(* PLC project sample_project, sample_company sample_product 1 *)
(* stored: creationDateTime 2024-07-18T21:30:47, modificationDateTime 2024-07-18T22:03:54 *)

FUNCTION_BLOCK sample_function_block_FBD
  VAR_INPUT
    Reset : BOOL;
  END_VAR
  VAR_OUTPUT
    Out : INT;
  END_VAR
  VAR
    Cnt : INT;
  END_VAR
  VAR_EXTERNAL CONSTANT
    ResetCounterValue : INT;
  END_VAR
  VAR  (* added by the conversion: wires and edge detectors of the diagram *)
    _SEL4_OUT : ANY;
  END_VAR

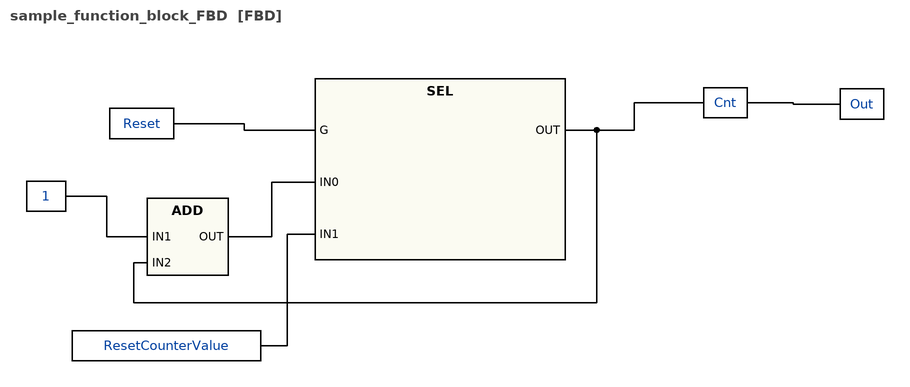
(* FBD diagram, written out as Structured Text *)
Out := Cnt;
_SEL4_OUT := SEL(Reset, 1 + _SEL4_OUT, ResetCounterValue);
Cnt := _SEL4_OUT;
END_FUNCTION_BLOCK

(* Counter in ST language *)
FUNCTION_BLOCK sample_function_block_ST
  VAR_INPUT
    Reset : BOOL;
  END_VAR
  VAR_OUTPUT
    Out : INT;
  END_VAR
  VAR
    Cnt : INT;
  END_VAR
  VAR_EXTERNAL CONSTANT
    ResetCounterValue : INT;
  END_VAR

            IF Reset THEN
  Cnt := ResetCounterValue;
ELSE
  Cnt := Cnt + 1;
END_IF;

Out := Cnt;
          
END_FUNCTION_BLOCK

PROGRAM sample_program
  VAR_INPUT
    Reset : BOOL;
  END_VAR
  VAR_OUTPUT
    Cnt0 : INT;
    Cnt1 : INT;
    Cnt2 : INT;
    Cnt3 : INT;
    Cnt4 : INT;
  END_VAR
  VAR
    sample_function_block_ST0 : sample_function_block_ST;
    sample_function_block_FBD0 : sample_function_block_FBD;
  END_VAR

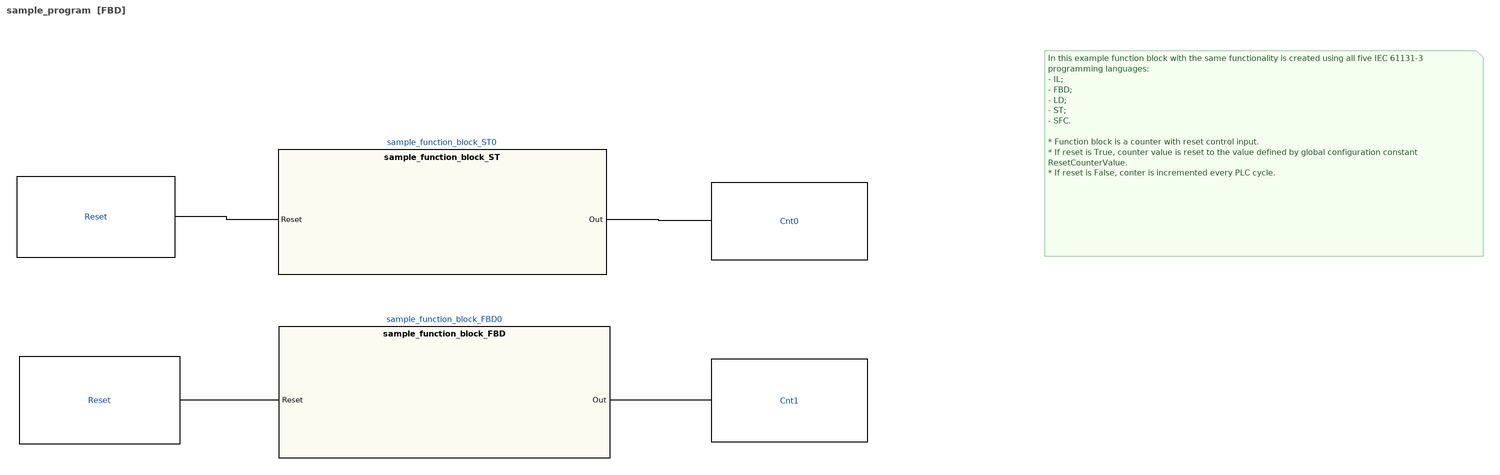
(* FBD diagram, written out as Structured Text *)
(* In this example function block with the same functionality is created using all five IEC 61131-3 programming languages:
- IL;
- FBD;
- LD;
- ST;
- SFC.

* Function block is a counter with reset control input.
* If reset is True, counter value is reset to the value defined by global configuration constant ResetCounterValue.
* If reset is False, conter is incremented every PLC cycle. *)
sample_function_block_ST0(Reset := Reset);
Cnt0 := sample_function_block_ST0.Out;
sample_function_block_FBD0(Reset := Reset);
Cnt1 := sample_function_block_FBD0.Out;
END_PROGRAM

CONFIGURATION sample_config
  VAR_GLOBAL CONSTANT
    ResetCounterValue : INT := 17;
  END_VAR
  RESOURCE sample_resource ON PLC
    TASK sample_task(INTERVAL := T#200ms, PRIORITY := 0);
    PROGRAM sample_task_instance WITH sample_task : sample_program;
  END_RESOURCE
END_CONFIGURATION
